(* CODESYS project 2019-07-30 Thingsboard  Subscribe.ecp

Project tree, tasks and I/O mapping:
  PFC_Sub : 750-8212 PFC200 2ETH RS, WAGO, order no. 0750-8212, version 5.13.2.32
    application Application
      libraries: ; VisuDialogs, * (System); WagoAppCloud, 1.3.0.7 (WAGO); WagoAppJSON, 1.0.1.1 (WAGO)
      task PLC_Task (cyclic, interval 100 ms, priority 15) calls PLC_PRG
      task VISU_TASK (cyclic, interval 100 ms, priority 15) calls VisuElems.Visu_Prg
      program PLC_PRG [ST]
      01_Cloud/
        program JSON_Converter [ST]
        program NativeMQTT_Subscribe [ST]
      visualisation Visualization
      global variables GVL
      data type BrokerConfig
      data type topicList
    Common.PCI
    Kbus : Kbus, WAGO, version 1.4.0.2
        unmapped channels: K-BUS diagnostics
    MODBUS
      MODBUS : MODBUS, WAGO, order no. n/a, version 1.1.1.15
    Serial
      COM1 : COM1, WAGO, version 0.0.0.19
  libraries: VisuSymbols, 3.5.10.0 (System); WagoVisuIcons, 1.0.1.0 (WAGO)
  text list GlobalTextList
  5ce3da45-db07-42e7-a21c-a00fff4ed8f6|Bilder\Lupe.PNG
  5ce3da45-db07-42e7-a21c-a00fff4ed8f6|Bilder\WAGO_2017_SPS_Messe_Saftfabrik_Freigestellt.png
  5ce3da45-db07-42e7-a21c-a00fff4ed8f6|Bilder\Tank_00_0398.png
  5ce3da45-db07-42e7-a21c-a00fff4ed8f6|Bilder\Tank_10_0398.png
  5ce3da45-db07-42e7-a21c-a00fff4ed8f6|Bilder\Tank_20_0398.png
  5ce3da45-db07-42e7-a21c-a00fff4ed8f6|Bilder\Tank_30_0398.png
  5ce3da45-db07-42e7-a21c-a00fff4ed8f6|Bilder\Tank_40_0398.png
  5ce3da45-db07-42e7-a21c-a00fff4ed8f6|Bilder\Tank_50_0398.png
  5ce3da45-db07-42e7-a21c-a00fff4ed8f6|Bilder\Tank_60_0398.png
  5ce3da45-db07-42e7-a21c-a00fff4ed8f6|Bilder\Tank_70_0398.png
  5ce3da45-db07-42e7-a21c-a00fff4ed8f6|Bilder\Tank_80_0398.png
  5ce3da45-db07-42e7-a21c-a00fff4ed8f6|Bilder\Tank_90_0398.png
  5ce3da45-db07-42e7-a21c-a00fff4ed8f6|Bilder\Tank_100_0398.png
*)

// PFC_Sub/Application/BrokerConfig
TYPE BrokerConfig :
STRUCT
	name:STRING:='';		//Name of the MQTT Broker
	pubTopic:STRING:='';	// Public topic
	subTopic:STRING:='';	// Subscribe topic
	myTemplateString:STRING(1000):='';//Template String for JSON conversion JSON library required
END_STRUCT
END_TYPE

// PFC_Sub/Application/topicList
TYPE topicList :
STRUCT
	topic:STRING:='';
	subscribed:BOOL:=FALSE;
	payload:STRING(256):='';
	subData	: ARRAY [0..254] OF BYTE;
END_STRUCT
END_TYPE

// PFC_Sub/Application/GVL
{attribute 'qualified_only'}
VAR_GLOBAL
	myPubTopic:STRING:='topic_0';	//Publish topic from visu
	myPubToggle:BOOL:=FALSE;//Toglle flag to trigger a new publish
	
	// 3 publish variables
	myPubString:STRING:='';	//Publish var 1 as String
	myPubInt:INT:=0;
	myPubReal:REAL:=0;
	
	mySubTopic:STRING:='';			// Topic for subscription
	mySubString:STRING(256):='';	// Buffer for subscribe payload
		
	MySubFlag:BOOL:=FALSE;	//Subscribe / unsubscribe flag
	
	myTemplateString:STRING(1000):='';//Template String for JSON library
END_VAR

// PFC_Sub/Application/PLC_PRG
PROGRAM PLC_PRG
VAR
	myOldText:STRING:='';
	myOldInt:INT:=0;
	myOldReal:REAL:=0;
	dwCycleCount		: INT := 0;	
	
	textList1:ARRAY[0..1,0..24]OF STRING;
	textList2:ARRAY[0..1,25..49]OF STRING;
	subsribedList1:ARRAY[0..24]OF BOOL;
	subsribedList2:ARRAY[25..49]OF BOOL;
	
	i: INT:=0;
	topic:STRING:='PFC_';
END_VAR

dwCycleCount:=dwCycleCount+1;

//GVL.myPubTopic:='topic_0';	//topic specified by thingsboard
GVL.mySubTopic:='v1/devices/me/attributes';	//topic specified by thingsboard
GVL.myTemplateString:='{"myText": "#Parameter","myInt": "#Parameter","myReal": "#Parameter"}'; //Thingsboard.io

IF(myOldText <> GVL.myPubString) OR (myOldInt <> GVL.myPubInt) OR (myOldReal <> GVL.myPubReal)THEN
	GVL.myPubToggle:=TRUE;
	myOldText:=GVL.myPubString;
	myOldInt:=GVL.myPubInt;
	myOldReal:=GVL.myPubReal;
ELSE
	GVL.myPubToggle:=FALSE;
END_IF

NativeMQTT_Subscribe();

FOR i := 0 TO 24 BY 1 DO
	textList1[0,i]:=NativeMQTT_Subscribe.myTopicList[i].topic;
	textList1[1,i]:=NativeMQTT_Subscribe.myTopicList[i].payload;
	subsribedList1[i] := NativeMQTT_Subscribe.myTopicList[i].subscribed;
END_FOR;
FOR i := 25 TO 49 BY 1 DO
	textList2[0,i]:=NativeMQTT_Subscribe.myTopicList[i].topic;
	textList2[1,i]:=NativeMQTT_Subscribe.myTopicList[i].payload;
	subsribedList2[i] := NativeMQTT_Subscribe.myTopicList[i].subscribed;
END_FOR;

END_PROGRAM

// PFC_Sub/Application/01_Cloud/NativeMQTT_Subscribe
PROGRAM NativeMQTT_Subscribe

VAR
	dwCycleCount		: DWORD := 0;	

	mySubscribers : ARRAY[0..50] OF WagoAppCloud.FbSubscribeMQTT;
	myTopicList:ARRAY[0..50] OF topicList;

	i:INT:=0;
	init:BOOL:=TRUE;
END_VAR

dwCycleCount := dwCycleCount + 1;

IF (init=TRUE) THEN
	init:=FALSE;
	FOR i := 0 TO 49 BY 1 DO
		myTopicList[i].topic:=CONCAT('topic_',INT_TO_STRING(i));
	END_FOR;
END_IF

IF dwCycleCount>1 THEN
	FOR i := 0 TO 49 BY 1 DO
		mySubscribers[i](xSubscribe := TRUE, sTopic := myTopicList[i].topic, eQoS := eQualityOfService.QoS1, aPayloadData:= myTopicList[i].subData); 
		MemCopySecure(pDest:= ADR(myTopicList[i].payload), udiDestSize:= 255, pSource:= ADR(myTopicList[i].subData), udiSourceSize:= mySubscribers[i].dwRxNBytes, bPadding:= 0);

		IF myTopicList[i].payload<>'' THEN
			myTopicList[i].subscribed:=TRUE;
			
		END_IF
	END_FOR;	
END_IF

END_PROGRAM

// PFC_Sub/Application/01_Cloud/JSON_Converter
PROGRAM JSON_Converter
VAR_INPUT
	value1:STRING:='';
	value2:INT:=0;
	value3:REAL:=0;
	trigger:BOOL:=TRUE;
END_VAR
VAR
	fbjson: WagoAppJSON.Fb_JSON_Writer_01;
	
	MyTemplateString :STRING(1000) := '';
	MyValueArray: ARRAY [0..2] OF STRING;
	xTrig: BOOL := TRUE;
	sOutput: STRING(JSON_MAX_STRING);
END_VAR

MyValueArray[0]:=value1;
MyValueArray[1]:=TO_STRING(value2);
MyValueArray[2]:=TO_STRING(value3);

MyTemplateString:=GVL.myTemplateString;
fbjson(
	sJSON_BaseFrame:= MyTemplateString,
	oStatus=> , 
	xError=> , 
	xDone=> , 
	aParameterValues:= MyValueArray, 
	xTrigger:= trigger, 
	sOutput:= sOutput);

END_PROGRAM

// PFC_Sub/Application/Visualization
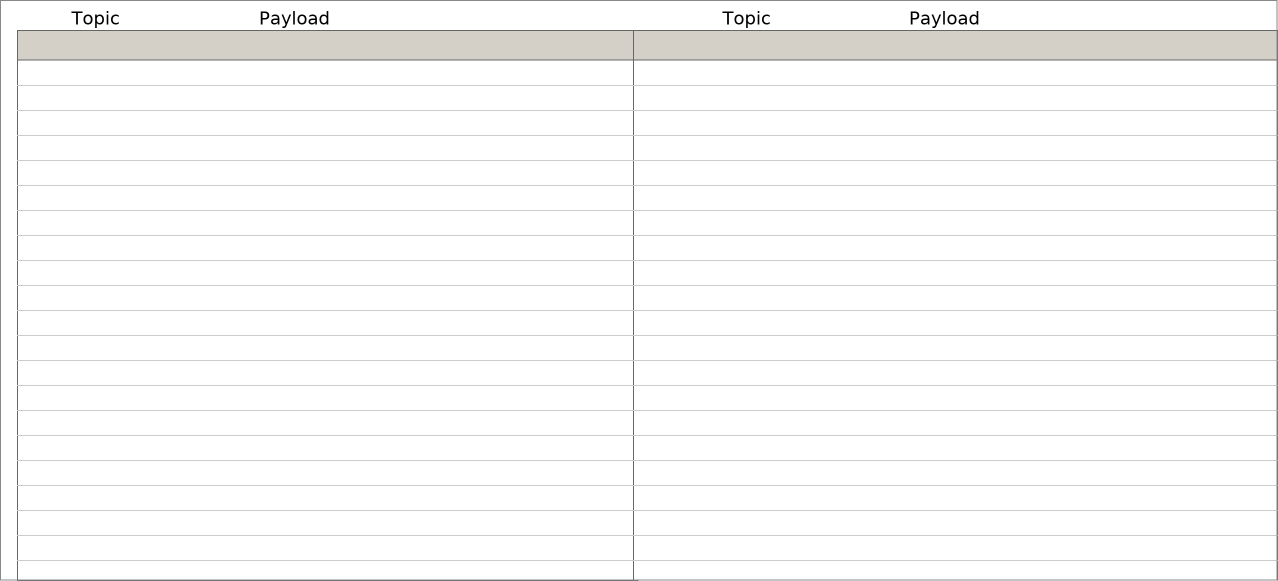
VISUALIZATION Visualization  // 1278x581
    Table (17,30 621x551), data array: PLC_PRG.textList1
        p3854506369: PLC_PRG.textList1[0,INDEX]
        p1892666644: PLC_PRG.textList1[1,INDEX]
    Table (633,30 645x550), data array: PLC_PRG.textList2
        p3854506369: PLC_PRG.textList2[0,INDEX]
        p1892666644: PLC_PRG.textList2[1,INDEX]
    Label (61,9 70x19), "Topic"
    Label (170,9 249x19), "Payload"
    Label (820,9 249x19), "Payload"
    Label (712,9 70x19), "Topic"
END_VISUALIZATION
